// Mitsubishi GX Works2 project: PLC_GROUP17_3   PLC: FX3G

// global labels: Global1
VAR_GLOBAL
  Start_Day AT X007 : BOOL;
  Emergency AT X005 : BOOL;
  Working_Day AT M1 : BOOL;
  Out_Of_Material AT M5 : BOOL;
  L_Work AT Y000 : BOOL;
  Oat_Amount AT D1100 : INT;
  Oat_Container AT D1105 : INT;
  Protein_Amount AT D1110 : INT;
  Protein_Countainer AT D1115 : INT;
  Honey_Amount AT D1120 : INT;
  Honey_Container AT D1125 : INT;
  Start_Mixing AT X003 : BOOL;
  Mixing_Timer AT TC1 : BOOL;
END_VAR
VAR_GLOBAL CONSTANT
  CONST5 : REAL := 5.0;
END_VAR
VAR_GLOBAL
  Mixing_Light AT Y003 : BOOL;
END_VAR
VAR_GLOBAL CONSTANT
  CONST6 : REAL := 6.0;
END_VAR
VAR_GLOBAL
  ProtainSnack AT M17 : BOOL;
END_VAR
VAR_GLOBAL CONSTANT
  CONST10 : REAL := 10;
END_VAR
VAR_GLOBAL
  ClassicSnack AT M18 : BOOL;
END_VAR
VAR_GLOBAL CONSTANT
  CONST50 : INT := 50;
  CONST400 : INT := 400;
END_VAR
VAR_GLOBAL
  SnackType AT D1205 : REAL;
  AnalogInput1 AT D8280 : INT;
  MixingTime AT TS1 : BOOL;
END_VAR
VAR_GLOBAL CONSTANT
  CONST_400 : REAL := 400.0;
  CONST_320 : REAL := 320.0;
  CONST_160 : REAL := 160.0;
  CONST_240 : REAL := 240.0;
  CONST_120 : REAL := 120.0;
END_VAR
VAR_GLOBAL
  Start_Bake AT X002 : BOOL;
  Working_Mixing AT M3 : BOOL;
  End_Mixing AT M14 : BOOL;
  OatContainer AT D1140 : REAL;
  ProteinContainer AT D1145 : REAL;
  HoneyContainer AT D1150 : REAL;
  Out_Put AT D8282 : INT;
  End_Of_Day AT M16 : BOOL;
  Working_Bake AT M24 : BOOL;
  End_Bake AT M26 : BOOL;
  Bake_Classic_Timer AT TC2 : BOOL;
END_VAR
VAR_GLOBAL CONSTANT
  CONST40 : INT := 40;
END_VAR
VAR_GLOBAL
  Bake_Protain_Timer AT TC3 : BOOL;
  Bake_Classic_Time AT TS2 : BOOL;
  Bake_Protain_Time AT TS3 : BOOL;
  Working_Bake_Light AT M27 : BOOL;
  Flashing_Lights_Timer AT TC5 : BOOL;
  Flashing_Light1_Timer AT TC5 : BOOL;
  Flashing_Light2_Timer AT TC6 : BOOL;
  Flashing_Light1 AT Y001 : BOOL;
END_VAR
VAR_GLOBAL CONSTANT
  CONST30 : INT := 30;
END_VAR
VAR_GLOBAL
  Flashing_Light2 AT Y002 : BOOL;
  Flashing_Light2_Time AT TS6 : BOOL;
  Flashing_Lights_Control AT M28 : BOOL;
  Start_Packing AT X006 : BOOL;
  Working_Packing AT M29 : BOOL;
  End_Packing AT M30 : BOOL;
  MixingCountainer AT D1170 : REAL;
END_VAR
VAR_GLOBAL CONSTANT
  CONST_680 : REAL := 680.00;
  CONST_720 : REAL := 720.00;
END_VAR
VAR_GLOBAL
  Produce_Snack AT X000 : BOOL;
  Snack_Counter AT CC1 : BOOL;
END_VAR
VAR_GLOBAL CONSTANT
  CONST7 : INT := 7;
END_VAR
VAR_GLOBAL
  SnackCounter AT CS1 : BOOL;
  Snack_Packaging_Light AT Y004 : BOOL;
  SnackCounterStatus AT CN1 : INT;
END_VAR
VAR_GLOBAL CONSTANT
  CONST1 : INT := 1;
  CONST_6 : INT := 6;
END_VAR
VAR_GLOBAL
  SnacksStorage AT D1190 : REAL;
END_VAR
VAR_GLOBAL CONSTANT
  CONST_1 : REAL := 1;
END_VAR
VAR_GLOBAL
  Daily_Amount_Output AT D1300 : REAL;
  End_Of_Workday AT M32 : BOOL;
  BakeCountainer AT D1270 : REAL;
  Flashing_Light1_Time AT TS5 : BOOL;
  Pack_light AT M40 : BOOL;
  Stop_Light_Pack AT M50 : BOOL;
END_VAR
VAR_GLOBAL CONSTANT
  CONST8 : INT := 8;
END_VAR
VAR_GLOBAL
  Tayp_Protain AT M57 : BOOL;
  Tayp_Classic AT M58 : BOOL;
  New_Day AT M61 : BOOL;
END_VAR
VAR_GLOBAL CONSTANT
  CONST_399 : REAL := 399.0;
  CONST_319 : REAL := 319.0;
  CONST_159 : REAL := 159.0;
END_VAR

// task Task_01 (event TRUE, interval 0, priority 31): POU_01

PROGRAM POU_01
(* structured ladder/FBD written out as ST: instructions are called as NAME(EN, inputs, outputs); _pN, _eN, _tN stand for wires *)
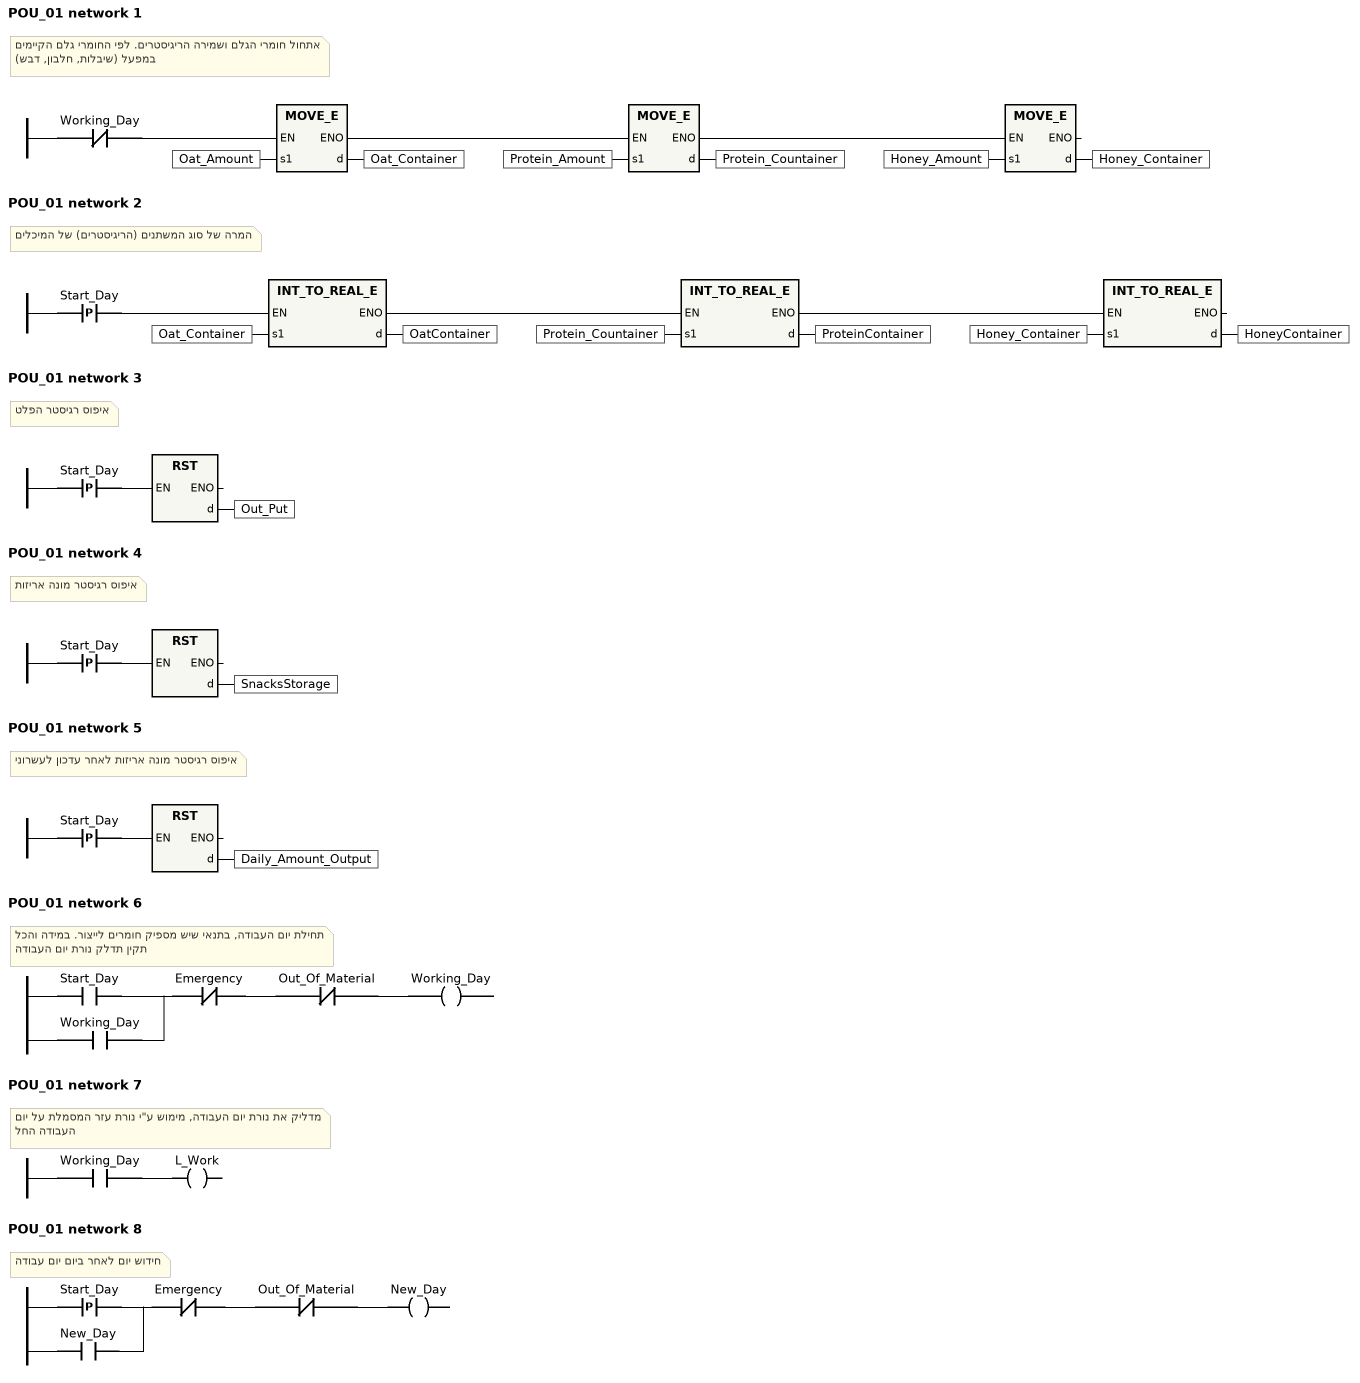
(* network 1 *)
(* אתחול חומרי הגלם ושמירה הריגיסטרים. לפי החומרי גלם הקיימים  במפעל (שיבלות, חלבון, דבש) *)
_e1 := MOVE_E(NOT Working_Day, Oat_Amount, Oat_Container);
_e2 := MOVE_E(_e1, Protein_Amount, Protein_Countainer);
MOVE_E(_e2, Honey_Amount, Honey_Container);
(* network 2 *)
(* המרה של סוג המשתנים (הריגיסטרים) של המיכלים *)
_e1 := INT_TO_REAL_E(LDP(TRUE, Start_Day), Oat_Container, OatContainer);
_e2 := INT_TO_REAL_E(_e1, Protein_Countainer, ProteinContainer);
INT_TO_REAL_E(_e2, Honey_Container, HoneyContainer);
(* network 3 *)
(* איפוס רגיסטר הפלט *)
RST(LDP(TRUE, Start_Day), Out_Put);
(* network 4 *)
(* איפוס רגיסטר מונה אריזות *)
RST(LDP(TRUE, Start_Day), SnacksStorage);
(* network 5 *)
(* איפוס רגיסטר מונה אריזות לאחר עדכון לעשרוני *)
RST(LDP(TRUE, Start_Day), Daily_Amount_Output);
(* network 6 *)
(* תחילת יום העבודה, בתנאי שיש מספיק חומרים לייצור. במידה והכל תקין תדלק נורת יום העבודה *)
Working_Day := ((Start_Day OR Working_Day) AND NOT Emergency) AND NOT Out_Of_Material;
(* network 7 *)
(* מדליק את נורת יום העבודה, מימוש ע"י נורת עזר המסמלת על יום העבודה החל *)
L_Work := Working_Day;
(* network 8 *)
(* חידוש יום לאחר ביום יום עבודה *)
New_Day := ((LDP(TRUE, Start_Day) OR New_Day) AND NOT Emergency) AND NOT Out_Of_Material;
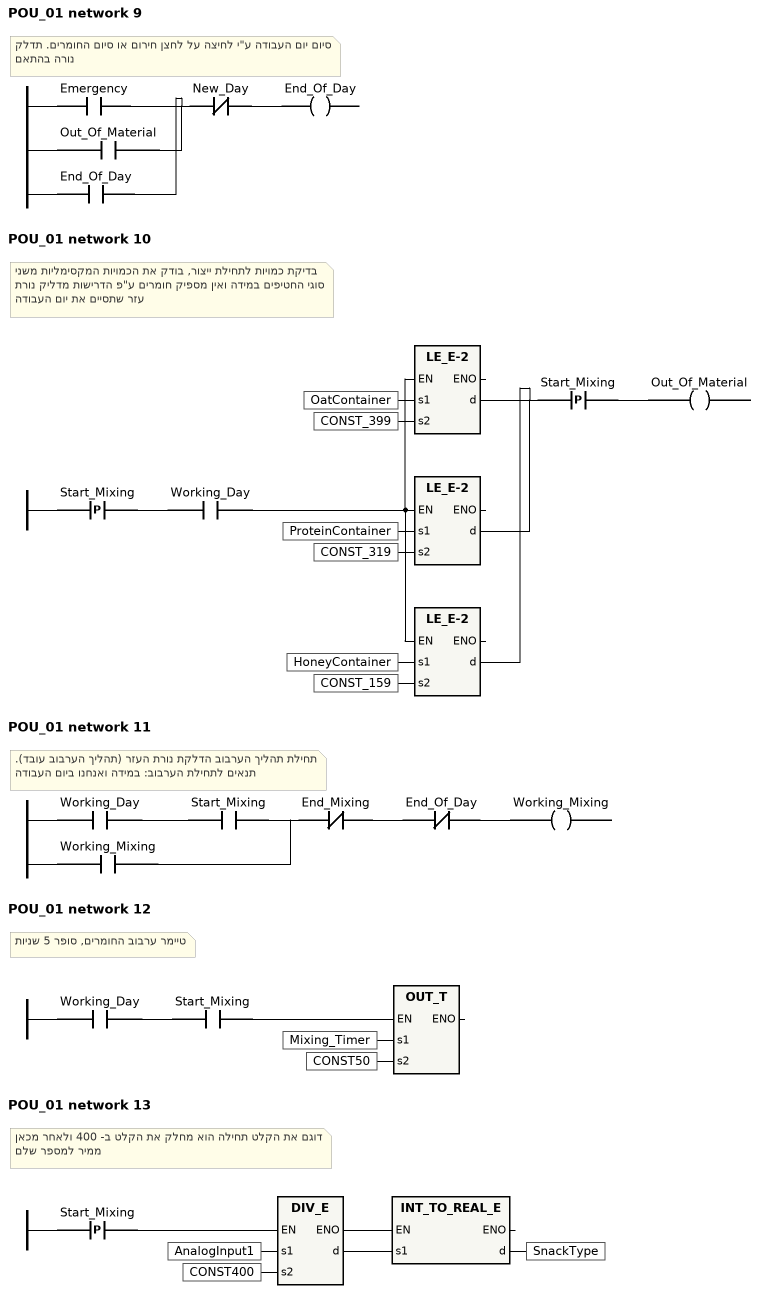
(* network 9 *)
(* סיום יום העבודה ע"י לחיצה על לחצן חירום או סיום החומרים. תדלק נורה בהתאם *)
End_Of_Day := (Emergency OR Out_Of_Material OR End_Of_Day) AND NOT New_Day;
(* network 10 *)
(* בדיקת כמויות לתחילת ייצור, בודק את הכמויות המקסימליות משני סוגי החטיפים במידה ואין מספיק חומרים ע"פ הדרישות מדליק נורת עזר שתסיים את יום העבודה *)
_p1 := LDP(TRUE, Start_Mixing) AND Working_Day;
LE_E(_p1, OatContainer, CONST_399, _t2);
LE_E(_p1, ProteinContainer, CONST_319, _t3);
LE_E(_p1, HoneyContainer, CONST_159, _t4);
Out_Of_Material := (_t2 OR _t3 OR _t4) AND LDP(TRUE, Start_Mixing);
(* network 11 *)
(* תחילת תהליך הערבוב הדלקת נורת העזר (תהליך הערבוב עובד). תנאים לתחילת הערבוב: במידה ואנחנו ביום העבודה *)
Working_Mixing := (((Working_Day AND Start_Mixing) OR Working_Mixing) AND NOT End_Mixing) AND NOT End_Of_Day;
(* network 12 *)
(* טיימר ערבוב החומרים, סופר 5 שניות *)
OUT_T(Working_Day AND Start_Mixing, Mixing_Timer, CONST50);
(* network 13 *)
(* דוגם את הקלט תחילה הוא מחלק את הקלט ב- 400 ולאחר מכאן ממיר למספר שלם *)
_e2 := DIV_E(LDP(TRUE, Start_Mixing), AnalogInput1, CONST400, _t1);
INT_TO_REAL_E(_e2, _t1, SnackType);
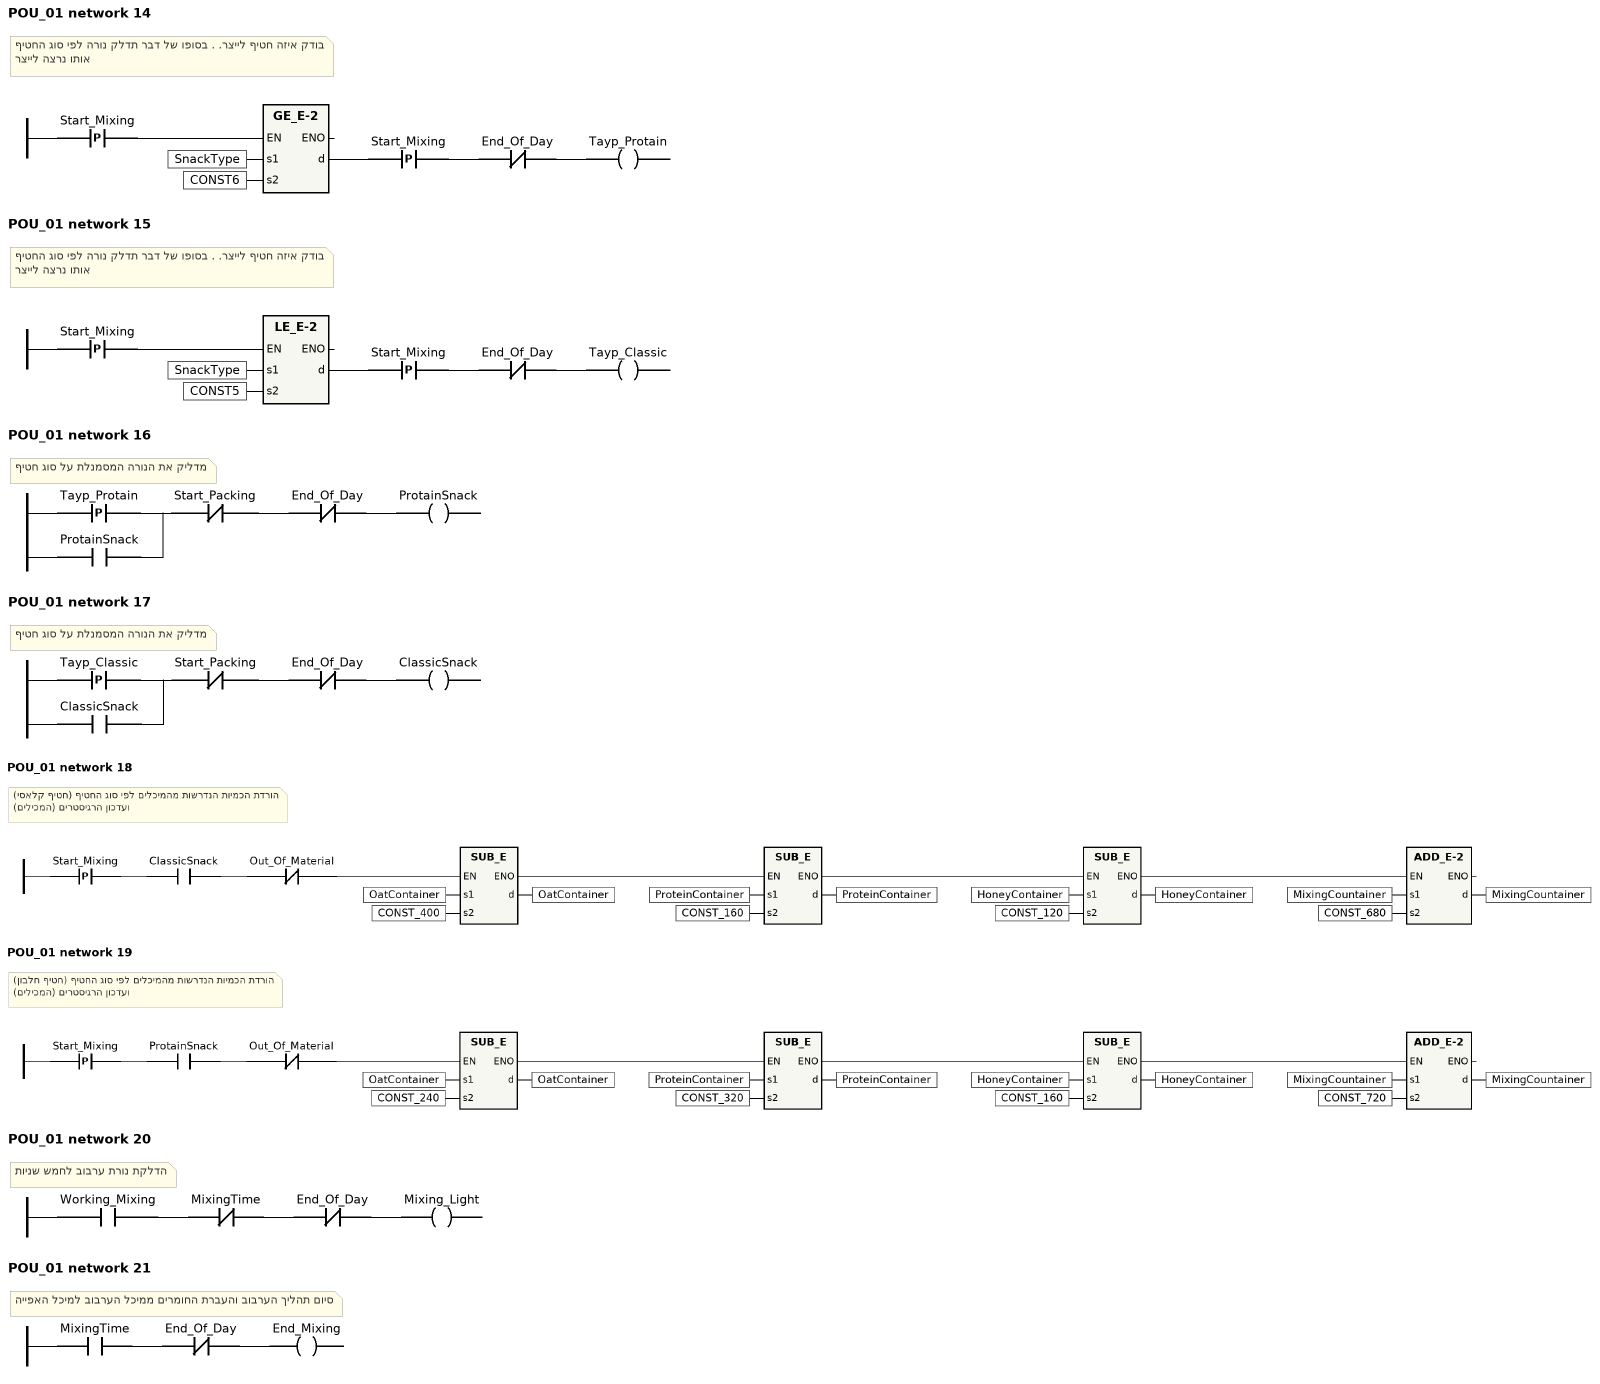
(* network 14 *)
(* בודק איזה חטיף לייצר. . בסופו של דבר תדלק נורה לפי סוג החטיף אותו נרצה לייצר *)
GE_E(LDP(TRUE, Start_Mixing), SnackType, CONST6, _t1);
Tayp_Protain := _t1 AND LDP(TRUE, Start_Mixing) AND NOT End_Of_Day;
(* network 15 *)
(* בודק איזה חטיף לייצר. . בסופו של דבר תדלק נורה לפי סוג החטיף אותו נרצה לייצר *)
LE_E(LDP(TRUE, Start_Mixing), SnackType, CONST5, _t1);
Tayp_Classic := _t1 AND LDP(TRUE, Start_Mixing) AND NOT End_Of_Day;
(* network 16 *)
(* מדליק את הנורה המסמנלת על סוג חטיף *)
ProtainSnack := ((LDP(TRUE, Tayp_Protain) OR ProtainSnack) AND NOT Start_Packing) AND NOT End_Of_Day;
(* network 17 *)
(* מדליק את הנורה המסמנלת על סוג חטיף *)
ClassicSnack := ((LDP(TRUE, Tayp_Classic) OR ClassicSnack) AND NOT Start_Packing) AND NOT End_Of_Day;
(* network 18 *)
(* הורדת הכמיות הנדרשות מהמיכלים לפי סוג החטיף (חטיף קלאסי) ועדכון הרגיסטרים (המכילים) *)
_e1 := SUB_E(LDP(TRUE, Start_Mixing) AND ClassicSnack AND NOT Out_Of_Material, OatContainer, CONST_400, OatContainer);
_e2 := SUB_E(_e1, ProteinContainer, CONST_160, ProteinContainer);
_e3 := SUB_E(_e2, HoneyContainer, CONST_120, HoneyContainer);
ADD_E(_e3, MixingCountainer, CONST_680, MixingCountainer);
(* network 19 *)
(* הורדת הכמיות הנדרשות מהמיכלים לפי סוג החטיף (חטיף חלבון) ועדכון הרגיסטרים (המכילים) *)
_e1 := SUB_E(LDP(TRUE, Start_Mixing) AND ProtainSnack AND NOT Out_Of_Material, OatContainer, CONST_240, OatContainer);
_e2 := SUB_E(_e1, ProteinContainer, CONST_320, ProteinContainer);
_e3 := SUB_E(_e2, HoneyContainer, CONST_160, HoneyContainer);
ADD_E(_e3, MixingCountainer, CONST_720, MixingCountainer);
(* network 20 *)
(* הדלקת נורת ערבוב לחמש שניות *)
Mixing_Light := Working_Mixing AND NOT MixingTime AND NOT End_Of_Day;
(* network 21 *)
(* סיום תהליך הערבוב והעברת החומרים ממיכל הערבוב למיכל האפייה *)
End_Mixing := MixingTime AND NOT End_Of_Day;
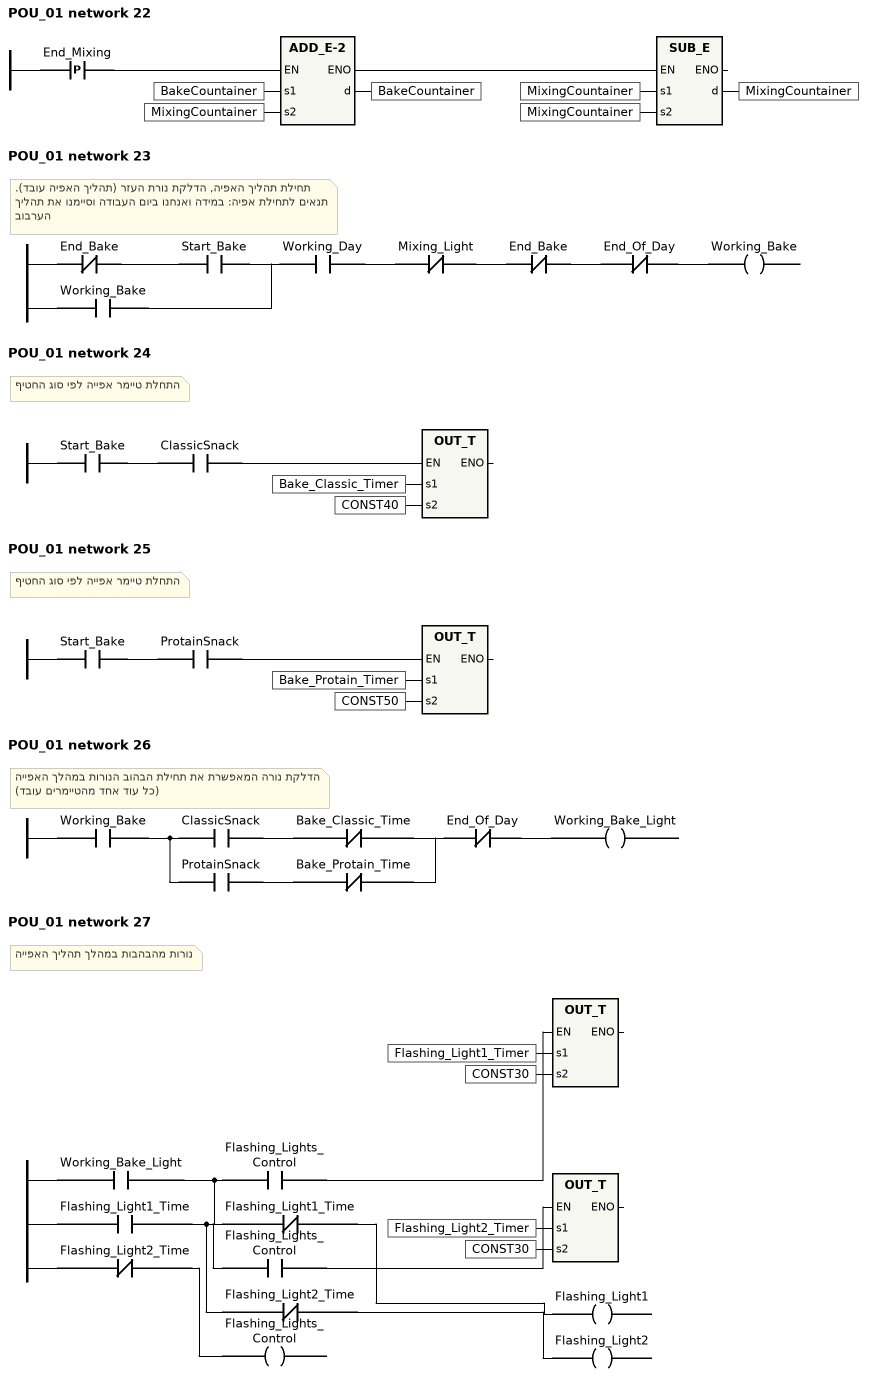
(* network 22 *)
_e1 := ADD_E(LDP(TRUE, End_Mixing), BakeCountainer, MixingCountainer, BakeCountainer);
SUB_E(_e1, MixingCountainer, MixingCountainer, MixingCountainer);
(* network 23 *)
(* תחילת תהליך האפיה, הדלקת נורת העזר (תהליך האפיה עובד). תנאים לתחילת אפיה: במידה ואנחנו ביום העבודה וסיימנו את תהליך הערבוב *)
Working_Bake := (((((NOT End_Bake AND Start_Bake) OR Working_Bake) AND Working_Day) AND NOT Mixing_Light) AND NOT End_Bake) AND NOT End_Of_Day;
(* network 24 *)
(* התחלת טיימר אפייה לפי סוג החטיף *)
OUT_T(Start_Bake AND ClassicSnack, Bake_Classic_Timer, CONST40);
(* network 25 *)
(* התחלת טיימר אפייה לפי סוג החטיף *)
OUT_T(Start_Bake AND ProtainSnack, Bake_Protain_Timer, CONST50);
(* network 26 *)
(* הדלקת נורה המאפשרת את תחילת הבהוב הנורות במהלך האפייה (כל עוד אחד מהטיימרים עובד) *)
Working_Bake_Light := ((Working_Bake AND ClassicSnack AND NOT Bake_Classic_Time) OR (Working_Bake AND ProtainSnack AND NOT Bake_Protain_Time)) AND NOT End_Of_Day;
(* network 27 *)
(* נורות מהבהבות במהלך תהליך האפייה *)
OUT_T(Working_Bake_Light AND Flashing_Lights_Control, Flashing_Light1_Timer, CONST30);
Flashing_Light1 := Working_Bake_Light AND NOT Flashing_Light1_Time;
OUT_T(Flashing_Light1_Time AND Flashing_Lights_Control, Flashing_Light2_Timer, CONST30);
Flashing_Light2 := Flashing_Light1_Time AND NOT Flashing_Light2_Time;
Flashing_Lights_Control := NOT Flashing_Light2_Time;
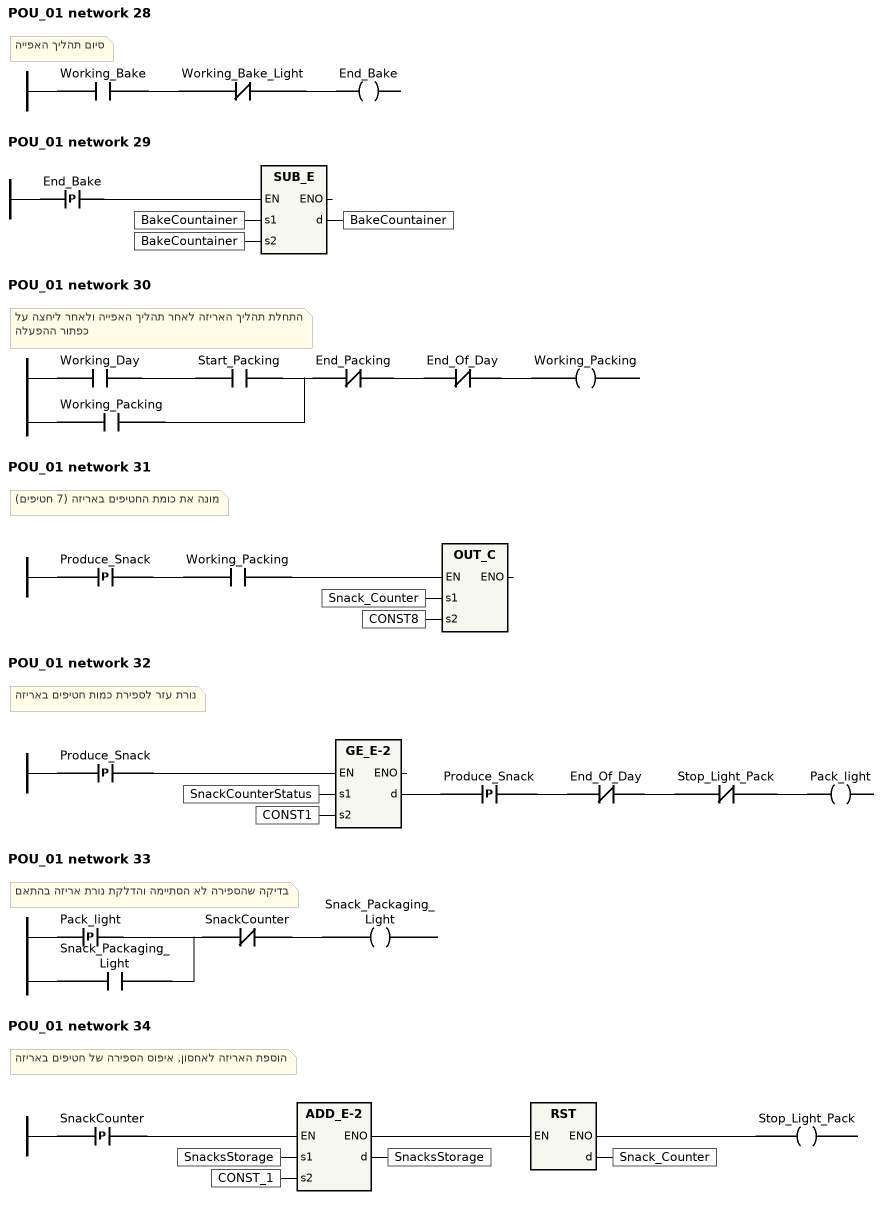
(* network 28 *)
(* סיום תהליך האפייה *)
End_Bake := Working_Bake AND NOT Working_Bake_Light;
(* network 29 *)
SUB_E(LDP(TRUE, End_Bake), BakeCountainer, BakeCountainer, BakeCountainer);
(* network 30 *)
(* התחלת תהליך האריזה לאחר תהליך האפייה ולאחר ליחצה על כפתור ההפעלה *)
Working_Packing := (((Working_Day AND Start_Packing) OR Working_Packing) AND NOT End_Packing) AND NOT End_Of_Day;
(* network 31 *)
(* מונה את כומת החטיפים באריזה (7 חטיפים) *)
OUT_C(LDP(TRUE, Produce_Snack) AND Working_Packing, Snack_Counter, CONST8);
(* network 32 *)
(* נורת עזר לספירת כמות חטיפים באריזה *)
GE_E(LDP(TRUE, Produce_Snack), SnackCounterStatus, CONST1, _t1);
Pack_light := _t1 AND LDP(TRUE, Produce_Snack) AND NOT End_Of_Day AND NOT Stop_Light_Pack;
(* network 33 *)
(* בדיקה שהספירה לא הסתיימה והדלקת נורת אריזה בהתאם *)
Snack_Packaging_Light := (LDP(TRUE, Pack_light) OR Snack_Packaging_Light) AND NOT SnackCounter;
(* network 34 *)
(* הוספת האריזה לאחסון, איפוס הספירה של חטיפים באריזה *)
_e1 := ADD_E(LDP(TRUE, SnackCounter), SnacksStorage, CONST_1, SnacksStorage);
_e2 := RST(_e1, Snack_Counter);
Stop_Light_Pack := _e2;
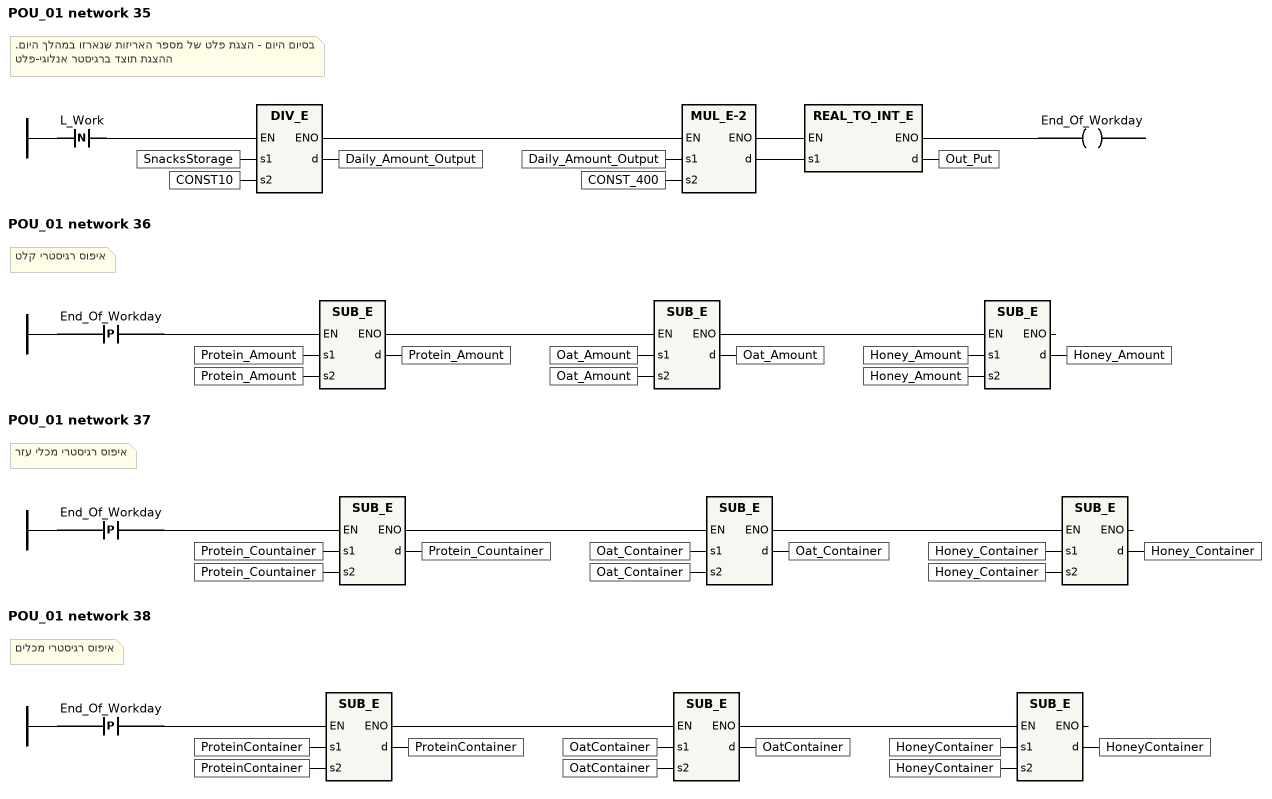
(* network 35 *)
(* בסיום היום - הצגת פלט של מספר האריזות שנארזו במהלך היום. ההצגת תוצד ברגיסטר אנלוגי-פלט *)
_e1 := DIV_E(LDF(TRUE, L_Work), SnacksStorage, CONST10, Daily_Amount_Output);
_e3 := MUL_E(_e1, Daily_Amount_Output, CONST_400, _t2);
_e4 := REAL_TO_INT_E(_e3, _t2, Out_Put);
End_Of_Workday := _e4;
(* network 36 *)
(* איפוס רגיסטרי קלט *)
_e1 := SUB_E(LDP(TRUE, End_Of_Workday), Protein_Amount, Protein_Amount, Protein_Amount);
_e2 := SUB_E(_e1, Oat_Amount, Oat_Amount, Oat_Amount);
SUB_E(_e2, Honey_Amount, Honey_Amount, Honey_Amount);
(* network 37 *)
(* איפוס רגיסטרי מכלי עזר *)
_e1 := SUB_E(LDP(TRUE, End_Of_Workday), Protein_Countainer, Protein_Countainer, Protein_Countainer);
_e2 := SUB_E(_e1, Oat_Container, Oat_Container, Oat_Container);
SUB_E(_e2, Honey_Container, Honey_Container, Honey_Container);
(* network 38 *)
(* איפוס רגיסטרי מכלים *)
_e1 := SUB_E(LDP(TRUE, End_Of_Workday), ProteinContainer, ProteinContainer, ProteinContainer);
_e2 := SUB_E(_e1, OatContainer, OatContainer, OatContainer);
SUB_E(_e2, HoneyContainer, HoneyContainer, HoneyContainer);
END_PROGRAM
